PROGRAM AxisEnable
VAR
END_VAR

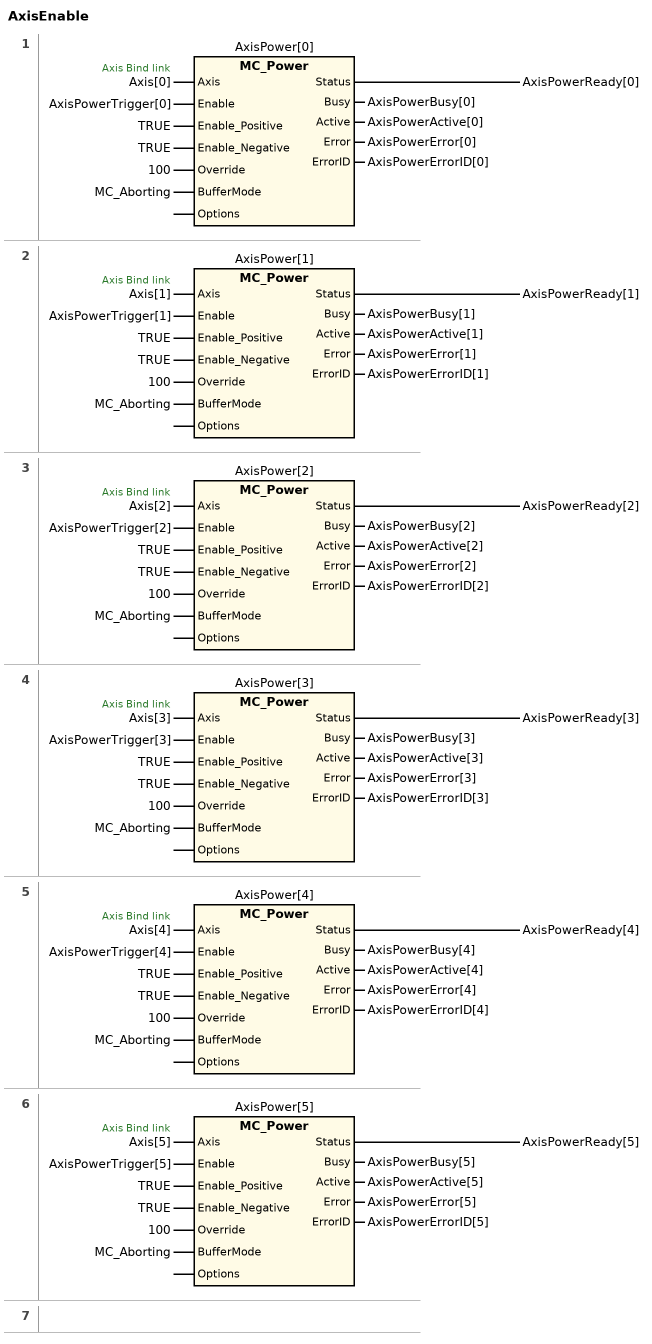
// NETWORK 1
//   AxisPower[0]: Axis Power On
//   Axis[0]: Axis Bind link
AxisPower[0](
    Axis := Axis[0],
    Enable := AxisPowerTrigger[0],
    Enable_Positive := TRUE,
    Enable_Negative := TRUE,
    Override := 100,
    BufferMode := MC_Aborting,
    Busy => AxisPowerBusy[0],
    Active => AxisPowerActive[0],
    Error => AxisPowerError[0],
    ErrorID => AxisPowerErrorID[0]); // MC_Power
AxisPowerReady[0] := AxisPower[0].Status;

// NETWORK 2
//   AxisPower[1]: Axis Power On
//   Axis[1]: Axis Bind link
AxisPower[1](
    Axis := Axis[1],
    Enable := AxisPowerTrigger[1],
    Enable_Positive := TRUE,
    Enable_Negative := TRUE,
    Override := 100,
    BufferMode := MC_Aborting,
    Busy => AxisPowerBusy[1],
    Active => AxisPowerActive[1],
    Error => AxisPowerError[1],
    ErrorID => AxisPowerErrorID[1]); // MC_Power
AxisPowerReady[1] := AxisPower[1].Status;

// NETWORK 3
//   AxisPower[2]: Axis Power On
//   Axis[2]: Axis Bind link
AxisPower[2](
    Axis := Axis[2],
    Enable := AxisPowerTrigger[2],
    Enable_Positive := TRUE,
    Enable_Negative := TRUE,
    Override := 100,
    BufferMode := MC_Aborting,
    Busy => AxisPowerBusy[2],
    Active => AxisPowerActive[2],
    Error => AxisPowerError[2],
    ErrorID => AxisPowerErrorID[2]); // MC_Power
AxisPowerReady[2] := AxisPower[2].Status;

// NETWORK 4
//   AxisPower[3]: Axis Power On
//   Axis[3]: Axis Bind link
AxisPower[3](
    Axis := Axis[3],
    Enable := AxisPowerTrigger[3],
    Enable_Positive := TRUE,
    Enable_Negative := TRUE,
    Override := 100,
    BufferMode := MC_Aborting,
    Busy => AxisPowerBusy[3],
    Active => AxisPowerActive[3],
    Error => AxisPowerError[3],
    ErrorID => AxisPowerErrorID[3]); // MC_Power
AxisPowerReady[3] := AxisPower[3].Status;

// NETWORK 5
//   AxisPower[4]: Axis Power On
//   Axis[4]: Axis Bind link
AxisPower[4](
    Axis := Axis[4],
    Enable := AxisPowerTrigger[4],
    Enable_Positive := TRUE,
    Enable_Negative := TRUE,
    Override := 100,
    BufferMode := MC_Aborting,
    Busy => AxisPowerBusy[4],
    Active => AxisPowerActive[4],
    Error => AxisPowerError[4],
    ErrorID => AxisPowerErrorID[4]); // MC_Power
AxisPowerReady[4] := AxisPower[4].Status;

// NETWORK 6
//   AxisPower[5]: Axis Power On
//   Axis[5]: Axis Bind link
AxisPower[5](
    Axis := Axis[5],
    Enable := AxisPowerTrigger[5],
    Enable_Positive := TRUE,
    Enable_Negative := TRUE,
    Override := 100,
    BufferMode := MC_Aborting,
    Busy => AxisPowerBusy[5],
    Active => AxisPowerActive[5],
    Error => AxisPowerError[5],
    ErrorID => AxisPowerErrorID[5]); // MC_Power
AxisPowerReady[5] := AxisPower[5].Status;

// NETWORK 7

END_PROGRAM

(* stored: Version 1.1.0.1, ProductVersion 3.1.4018.5
   POU AxisEnable: Id {d000457b-2b51-4361-b53d-474aa75a2836}, SpecialFunc None *)
